{attribute 'analysis' := '-33'}
PROGRAM PRG_TcUnit
VAR
	fbTcunitExample : FB_TcUnitExample;
	fbNoSnappy		: FB_TcUnitWithoutSnappyExample;
END_VAR



TcUnit.RUN();

END_PROGRAM

(* stored: Version 1.1.0.1, ProductVersion 3.1.4026.18
   POU PRG_TcUnit: Id {bc2d77bc-f8be-4d06-b9a5-5cd2e5ed9256}, SpecialFunc None *)
